// TIA Portal V17 export
// export: Created 2025-11-18T11:18:45.9396835Z, ExportSetting WithDefaults, DisplayName Totally Integrated Automation Portal, DisplayVersion V17 Update 8, DisplayName TIA Portal Openness, DisplayVersion V17 Update 8, DisplayName TIA Portal Version Control Interface, DisplayVersion V17, DisplayName STEP 7 Professional, DisplayVersion V17 Update 8, DisplayName STEP 7 Safety, DisplayVersion V17 Update 6, DisplayName WinCC Advanced, DisplayVersion V17 Update 8
DATA_BLOCK "PLC_VLC_DATA"   // DB11
{ S7_Optimized_Access := 'FALSE' }
VERSION : 0.1
// stored: AutoNumber true, DBAccessibleFromOPCUA true, IsOnlyStoredInLoadMemory false, IsWriteProtectedInAS false
   VAR
      Command : Struct
         Start : Bool;
         Stop : Bool;
         Reset : Bool;
         Pause : Bool;
         Resume : Bool;
         Rewind0 : Bool;
         RewindX : Bool;
      END_STRUCT;
      Status : Struct
         xConnected : Bool;
         xHeartbeat : Bool;
         xStarted : Bool;
         xPaused : Bool;
         xEndOfFile : Bool;
         xConnected_Memo : Bool;
         xStarted_Memo : Bool;
         xPaused_Memo : Bool;
         xEndOfFile_Memo : Bool;
         xConnectionOK : Bool;
      END_STRUCT;
      Requests : Struct
         xSendRequest : Bool;
         xDataReceiveOn : Bool := True;
         xReconnect : Bool;
         xRepeatInLoop : Bool := False;
         xStartAfterStopCondition : Bool;
      END_STRUCT;
      "Repeat" : Struct
         StartAgain : Bool;
         WaitForEnd : Bool;
         StopOnTheBegin : Bool;
         StartAfterStop : Bool;
         Rewind0AfterStopFirstCycle : Bool;
      END_STRUCT;
      Pulses : Array[0..10] of Bool;
   END_VAR
BEGIN
END_DATA_BLOCK
